// TIA Portal V20 export
TYPE "typeSequenceControlNodeInterafceSTK2"
// stored: Namespace Unit1.Em7
   STRUCT
      jobs { ExternalWritable := 'False'} : "LAF_typeJobs";
      sequence { ExternalWritable := 'False'} : "LAF_typeSequence";
      "step" { ExternalWritable := 'False'} : "LER_typeStep";
      jobInterface { ExternalWritable := 'False'} : "Unit1.Em7.typeSequenceControlNodeInterafceSTKJobInterface";
   END_STRUCT;
END_TYPE
